FUNCTION FLOOR (* This is a rounding function which returns the biggest possible integer which is less or equal to X. *)
  (* Standard: 61499-1 *)
  (* Version 1.0, 2025-12-21, Franz Höpfinger *)
  PACKAGE OSCAT::Basic::POUs::Mathematical;
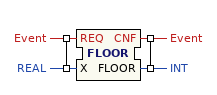
  EVENT_INPUT
    REQ WITH X;
  END_EVENT
  EVENT_OUTPUT
    CNF WITH FLOOR;
  END_EVENT
  VAR_INPUT
    X : REAL;
  END_VAR
  VAR_OUTPUT
    FLOOR : INT;
  END_VAR
  BODY IN ST:
PACKAGE OSCAT::Basic::POUs::Mathematical;

(* This is a rounding function which returns the biggest possible integer which is less or equal
 * to X. *)
FUNCTION FLOOR : INT
VAR_INPUT
	X : REAL;
END_VAR

(*
 * version 1.1	21. mar. 2008 programmer 	hugo tested by		tobias
 * *
 * This is a rounding function which returns the biggest possible integer which is less or equal to
 * X.
 * floor(3.14) = 3 floor(-3.14) = -4
 *)
FLOOR := REAL_TO_INT(X);
IF FLOOR > X THEN
	FLOOR := FLOOR - 1;
END_IF;

END_FUNCTION

(*
 * version 1.1	21. mar. 2008 programmer 	hugo tested by		tobias
 * *
 * This is a rounding function which returns the biggest possible integer which is less or equal to
 * X.
 * floor(3.14) = 3 floor(-3.14) = -4
 *)
  END_BODY
END_FUNCTION
